FUNCTION_BLOCK FbStirBlock IMPLEMENTS IStirBlock
VAR_INPUT
	
END_VAR
VAR_OUTPUT
	bStirBlockStarted: BOOL;
	bStirBlockEnded: BOOL;
	
END_VAR
VAR
	FbSimulator : fbSimulator;
	CurrentTarget: INT;

END_VAR

{warning 'add property implementation'}
PROPERTY pEndFeedback : BOOL
GET
pEndFeedback := bStirBlockEnded;
END_GET
END_PROPERTY

{warning 'add property implementation'}
PROPERTY pStartFeedback : BOOL
GET
pStartFeedback := bStirBlockStarted;
END_GET
END_PROPERTY

{warning 'add method implementation '}
METHOD Stir : BOOL
VAR_INPUT
	sTargetName : STRING;
	bStirStartCommand : BOOL;
	bStirEndCommand : BOOL;
	nStirSetPoint : INT;
END_VAR
VAR
END_VAR
IF sTargetName = 'RV_50L' THEN
	CurrentTarget := 1;
ELSIF  sTargetName = 'RV_25L' THEN
	CurrentTarget := 2;	
ELSIF  sTargetName = 'MVA' THEN
	CurrentTarget := 0;	
END_IF

IF nStirSetPoint <> 0 AND RecipeTags.bRecipeStatus THEN


	IF bStirStartCommand AND NOT(bStirEndCommand)THEN
		bStirBlockStarted := TRUE;
		IO.Reactors[CurrentTarget].VFD.nRPMSetPointScaled := nStirSetPoint;
	ELSE
		bStirBlockStarted := FALSE;
		IO.Reactors[CurrentTarget].VFD.nRPMSetPointScaled := 0;
	END_IF
ELSE
	bStirBlockStarted := FALSE;
END_IF

IO.Reactors[CurrentTarget].VFD.bStart := bStirBlockStarted;

IO.Reactors[CurrentTarget].VFD.nRPMSetPointScaled := nStirSetPoint;
//FbSimulator(CurrentValue := IO.Reactors[CurrentTarget].VFD.nRPMFeedBackScaled, TargetValue :=  nStirSetPoint,SimulatedValue => IO.Reactors[CurrentTarget].VFD.nRPMFeedBackScaled );

//	IF R1.RecipeStep[R1.StepCount].StirrerStartedTime = '' THEN
//		R1.RecipeStep[R1.StepCount].StirrerStartedTime := Main.concatenatedHourMinuteString;
//	END_IF

IF ABS(IO.Reactors[CurrentTarget].VFD.nRPMFeedBackScaled - nStirSetPoint)<= 5 THEN
	bStirBlockEnded := TRUE;	
//	IF R1.RecipeStep[R1.StepCount].StirrerEndedTime = '' THEN
//			R1.RecipeStep[R1.StepCount].StirrerEndedTime := Main.concatenatedHourMinuteString;
//		END_IF
ELSE 
		bStirBlockEnded := FALSE;	

END_IF

Stir := true;
END_METHOD

END_FUNCTION_BLOCK

(* stored: Version 1.1.0.1, ProductVersion 3.1.4024.5
   POU FbStirBlock: Id {d248f781-87bd-4dd5-a8fb-b266f7d526ef}, SpecialFunc None
   Property pEndFeedback: Id {23a29034-4c18-42e6-a6a6-521d1f79e941}
   Get Get: Id {8f07b5f0-423b-417e-95cc-b20cff45f624}
   Property pStartFeedback: Id {e83c7ec6-b3b8-43ba-8ea2-63faf54b561e}
   Get Get: Id {50e09bad-c4f5-433d-8549-a774c22315f6}
   Method Stir: Id {c5838d98-cc2d-43cf-94b4-56f833afffaf} *)
